FUNCTION_BLOCK FB_CNSystem EXTENDS FB_SystemContinous
VAR_INPUT
END_VAR
VAR_OUTPUT
END_VAR
VAR
	//pumps
	stPU196DefaultParameters : ST_PumpGrundfosMagna3DefaultParameters;
	PU196 : FB_PumpGrundfosMagna3 := (ST_DefaultParameters := stPU196DefaultParameters);
	
	//valves
	stSV196DefaultParameters : ST_DiscreteValveDefaultParameters;
	stSV197DefaultParameters : ST_DiscreteValveDefaultParameters;
	
	SV196 : FB_DiscreteValve := (ST_DefaultParameters := stSV196DefaultParameters);
	SV197 : FB_DiscreteValve := (ST_DefaultParameters := stSV197DefaultParameters);
	
	//sensors
	TVL196 : AutomationBaseClasses.FB_TemperatureSensor; //supply temperature cooling
	TRL196 : AutomationBaseClasses.FB_TemperatureSensor; //return temperature cooling
	
	WMZ196 : FB_MollineC3HeatCounter; //cooling network
	
	//internal variables
	bSetStatusOn_PU196 : BOOL;
	bSetStatusOn_SV196 : BOOL;
	bSetStatusOn_SV197 : BOOL;
	
	//clock
	bStartTimer : BOOL;
	Timer : TON;
	
END_VAR

Timer(IN := bStartTimer,
	PT := T#120S);
MAIN();

//pumps
PU196.GetState_Profibus();
PU196(bSetStatusOnAutomatic := bSetStatusOn_PU196,
	bAlgorithmPermission := bAlgorithmPermission,
	fSetPointAutomatic := fSetPoint,
	nControlModeAutomatic := 0);
PU196.SetState_Profibus();

//valves
SV196.GetState_BI();
SV196(bSetStatusOnAutomatic := bSetStatusOn_SV196,
	bAlgorithmPermission := bAlgorithmPermission);
SV196.SetState_BO();

SV197.GetState_BI();
SV197(bSetStatusOnAutomatic := bSetStatusOn_SV197,
	bAlgorithmPermission := bAlgorithmPermission);
SV197.SetState_BO();

//sensors
TVL196();
TVL196.GetState_AI();
TRL196();
TRL196.GetState_AI();

WMZ196(aHeatCounterTelegramm := MBus.Telegramm_WMZ_196);

METHOD PROTECTED  CheckError : BOOL
VAR_INPUT
END_VAR
VAR_OUTPUT
	bError : BOOL;
END_VAR
VAR
	bError_PU196 : BOOL;
END_VAR
bError := PU196.bError;
END_METHOD

METHOD PROTECTED  Operational : BOOL
VAR_INPUT
END_VAR
VAR_OUTPUT
	bSwitchToWorking : BOOL := FALSE;
END_VAR
bSetStatusOn_PU196 := TRUE;

IF PU196.bStatusOn THEN
	bSwitchToWorking := TRUE;
END_IF
END_METHOD

METHOD PROTECTED  RampDown : BOOL
VAR_INPUT
END_VAR
VAR_OUTPUT
	bRampDownFinished : BOOL := FALSE;
END_VAR
bSetStatusOn_PU196 := FALSE;

IF NOT PU196.bStatusOn THEN
	bSetStatusOn_SV196 := FALSE;
	bSetStatusOn_SV197 := FALSE;
	
	bStartTimer := TRUE;
	IF Timer.Q THEN
		bRampDownFinished := TRUE;
		bStartTimer := FALSE;
	END_IF
END_IF
END_METHOD

METHOD PROTECTED  RampUp : BOOL
VAR_INPUT
END_VAR
VAR_OUTPUT
	bRampUpFinished : BOOL := FALSE;
END_VAR
bSetStatusOn_SV196 := TRUE;
bSetStatusOn_SV197 := TRUE;

bStartTimer := TRUE;
IF Timer.Q THEN
	bStartTimer := FALSE;
	bRampUpFinished := TRUE;
END_IF
END_METHOD

METHOD PROTECTED   SetSetPointLimits : BOOL
VAR_INPUT
END_VAR
VAR_OUTPUT
END_VAR
aSetPointLimits[1] := 0;
aSetPointLimits[2] := 100;
END_METHOD

METHOD PROTECTED  SetState : BOOL
VAR_INPUT
END_VAR
VAR_OUTPUT
END_VAR
controlState.bStatusOn := bSetStatusOn;
setPointState.aSetPointLimits := aSetPointLimits;
setPointState.fSetPoint := fSetPoint;
setPointState.fOperatingPoint := fOperatingPoint;
setPointState.sSetPointUnit := 'percent';
setPointState.sOperatingPointUnit := 'percent';
END_METHOD

METHOD PROTECTED  Working : BOOL
VAR_INPUT
END_VAR
VAR_OUTPUT
	bSwitchToOperational : BOOL := FALSE;
END_VAR
//empty
END_METHOD

END_FUNCTION_BLOCK

(* stored: Version 1.1.0.1, ProductVersion 3.1.4024.6
   POU FB_CNSystem: Id {9062e5fc-34f5-40d1-9cf9-1141cc5ec15d}, SpecialFunc None
   Method CheckError: Id {cf393eb5-11e9-4ebf-9dae-c48e67d0e9eb}
   Method Operational: Id {56267dad-fec8-4e4e-a810-06a1491ea0b9}
   Method RampDown: Id {6beb78a7-0987-49fa-9a46-6426657e25a3}
   Method RampUp: Id {a7fff42e-0b7f-4dbc-9c67-408d61401906}
   Method SetSetPointLimits: Id {02a3828c-159c-458c-9549-b16532e710bd}
   Method SetState: Id {cdfab659-d11f-4eff-89da-750bdbacb162}
   Method Working: Id {7e04e338-6fab-4f22-ad0a-cbe669dbce2d} *)
